FUNCTION_BLOCK NeredaMetalSaltDosingLogic (* CAT Function Block Type *)
  (* Standard: 61499-2 *)
  (* Version 0.0, 7/9/2026, Schneider Electric, template *)
  PACKAGE SE.Nereda;
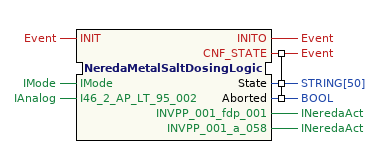
  EVENT_INPUT
    INIT;
  END_EVENT
  EVENT_OUTPUT
    INITO;
    CNF_STATE WITH State, Aborted;
  END_EVENT
  VAR_OUTPUT
    State : STRING[50];
    Aborted : BOOL;
  END_VAR
  SOCKETS
    IMode : IMode;
  END_SOCKETS
  SOCKETS
    I46_2_AP_LT_95_002 : IAnalog;
  END_SOCKETS
  PLUGS
    INVPP_001_fdp_001 : INeredaAct;
    INVPP_001_a_058 : INeredaAct;
  END_PLUGS
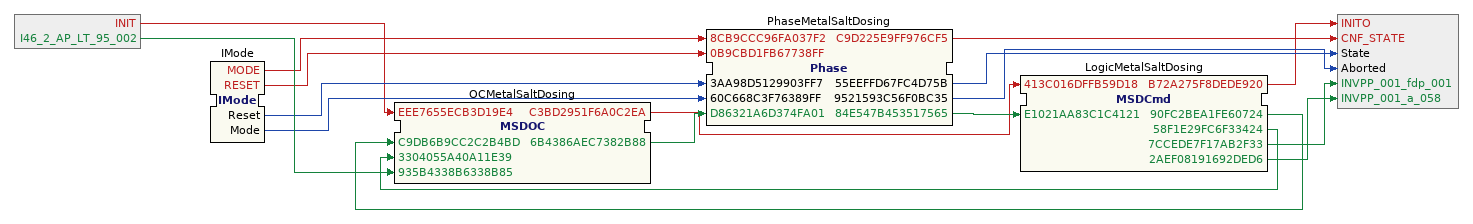
  (* 01 - FUNCTIONNAL INPUT INTERFACE *)
  (* 00 - INITIALIZATION *)
  (* 05 - LOGIC *)
  (* 06 - HMI INTERFACE *)
  (* 03 - FIELD INTERFACE *)
  (* Phase Feed *)
  (* 02 - FUNCTIONNAL OUTPUT INTERFACE *)
  FBS
    PhaseMetalSaltDosing : Phase;
    LogicMetalSaltDosing : MSDCmd;
    OCMetalSaltDosing : MSDOC;
  END_FBS
  EVENT_CONNECTIONS
    INIT TO OCMetalSaltDosing.EEE7655ECB3D19E4;
    OCMetalSaltDosing.C3BD2951F6A0C2EA TO LogicMetalSaltDosing.413C016DFFB59D18;
    LogicMetalSaltDosing.B72A275F8DEDE920 TO INITO;
    IMode.MODE TO PhaseMetalSaltDosing.8CB9CCC96FA037F2;
    IMode.RESET TO PhaseMetalSaltDosing.0B9CBD1FB67738FF;
    PhaseMetalSaltDosing.C9D225E9FF976CF5 TO CNF_STATE;
  END_CONNECTIONS
  DATA_CONNECTIONS
    IMode.Reset TO PhaseMetalSaltDosing.3AA98D5129903FF7;
    IMode.Mode TO PhaseMetalSaltDosing.60C668C3F76389FF;
    PhaseMetalSaltDosing.55EEFFD67FC4D75B TO State;
    PhaseMetalSaltDosing.9521593C56F0BC35 TO Aborted;
  END_CONNECTIONS
  ADAPTER_CONNECTIONS
    LogicMetalSaltDosing.90FC2BEA1FE60724 TO OCMetalSaltDosing.C9DB6B9CC2C2B4BD;
    LogicMetalSaltDosing.58F1E29FC6F33424 TO OCMetalSaltDosing.3304055A40A11E39;
    LogicMetalSaltDosing.7CCEDE7F17AB2F33 TO INVPP_001_fdp_001;
    LogicMetalSaltDosing.2AEF08191692DED6 TO INVPP_001_a_058;
    I46_2_AP_LT_95_002 TO OCMetalSaltDosing.935B4338B6338B85;
    PhaseMetalSaltDosing.84E547B453517565 TO LogicMetalSaltDosing.E1021AA83C1C4121;
    OCMetalSaltDosing.6B4386AEC7382B88 TO PhaseMetalSaltDosing.D86321A6D374FA01;
  END_CONNECTIONS
END_FUNCTION_BLOCK
